IF MlegRollBFinished=FALSE AND (gait_cycle-EnterMlegRollBCount)<=MlegRollBTime*gvl.sampleRate THEN
	body_ref_pos:=body_ref_pos_enter;
	body_ref_ang:=body_ref_ang_enter;
	leg_ref_pos:=leg_ref_pos_enter;
	tr  := UDINT_TO_LREAL(gait_cycle - EnterMlegRollBCount) / gvl.sampleRate / MlegRollBTime;
	fbGetPivot(tNow := tr, tTotal := 1.0, pivot => pvt);
	FOR i:=0 TO 1 DO
		FOR j:=0 TO 2 DO
			MlegRollB_MJntRef[i].data[j]:=(1-pvt)*MlegRollB_MJntStart[i].data[j]+pvt*(MlegRollB_MJntTarget[i,j]);
		END_FOR
		gvl.legCtrl[Mapping14[i]].ForwardKinetics(motorAngles:=MlegRollB_MJntRef[i].data , legIndex:=Mapping14[i] , tipPosition=>MlegRollB_MPosWrtHip[i].data );
		fbRotMat(yaw := body_ref_ang_enter.data[2], pitch := body_ref_ang_enter.data[1],roll := body_ref_ang_enter.data[0], rm =>  Rb_target1 );
		temp.data[0]:=hip_pos[Mapping14[i],0];temp.data[1]:=hip_pos[Mapping14[i],1];temp.data[2]:=hip_pos[Mapping14[i],2];
		leg_ref_pos[Mapping14[i]]:= VecAdd( MatMulVec(Rb_target1, VecAdd(temp,MatMulVec(Rleg[Mapping14[i]],MlegRollB_MPosWrtHip[i]))),body_ref_pos);
	END_FOR
	
	//force compensator
	tipForceTarget:=tipForceDesireLegAF;
	IF (gait_cycle-EnterMlegRollBCount)<=fceLoadTime*gvl.sampleRate THEN
		tr  := UDINT_TO_LREAL(gait_cycle-EnterMlegRollBCount) / gvl.sampleRate / fceLoadTime;
		fbGetPivot(tNow := tr, tTotal := 1.0, pivot => pvt);
		FOR i:=0 TO 5 DO
			FOR j:=0 TO 2 DO
				tipForceDesire[i,j]:=(1-pvt)*tipForceDesireZeros[i,j]+pvt*tipForceTarget[i,j];
			END_FOR
		END_FOR
	ELSIF (gait_cycle-EnterMlegRollBCount)>(MlegRollBTime-fceLoadTime)*gvl.sampleRate AND (gait_cycle-EnterMlegRollBCount)<=MlegRollBTime*gvl.sampleRate THEN
		tr  := (UDINT_TO_LREAL(gait_cycle-EnterMlegRollBCount) / gvl.sampleRate -(MlegRollBTime-fceLoadTime))/ fceLoadTime;
		fbGetPivot(tNow := tr, tTotal := 1.0, pivot => pvt);
		FOR i:=0 TO 5 DO
			FOR j:=0 TO 2 DO
				tipForceDesire[i,j]:=(1-pvt)*tipForceTarget[i,j]+pvt*tipForceDesireZeros[i,j];
			END_FOR
		END_FOR	
	END_IF	
	
ELSE	
	MlegRollBFinished:=TRUE;
	tipForceDesire:=tipForceDesireZeros;
END_IF
END_METHOD

METHOD PUBLIC TrjPlanning_MlegRollC : BOOL
VAR_INPUT
END_VAR
VAR
	MlegRollC_MPosTarget:ARRAY[0..1,0..2] OF LREAL:=[-0.2,-0.1797,-0.1246,
                                                     -0.2,-0.1797,0.1246];
	MlegRollC_MJntTargetRef:ARRAY[0..1,0..2] OF LREAL:=[0,523.2736*pi/180,-235.1052*pi/180,
                                                     0,523.2736*pi/180,-235.1052*pi/180];//invert rotation for shank and thigh, a more rotation for shank, old version										 
													 
	tr: lreal;
	i: INT;
	j: INT;
	Rb_target1: Mat3;
	temp: vec3;
	tempLeg:ARRAY [0..2] OF LREAL;
	tempJnt:ARRAY [0..2] OF LREAL;
	tempRef:ARRAY [0..2] OF LREAL;	
	
	tipForceDesireLegAF:	 ARRAY[0..5,0..2] OF LREAL:=[0,-100,0,
													 0,0,0,
													 0,0,0,
													 0,0,0,
													 0,0,0,
													 0,-120,0];
END_VAR
IF (gait_cycle-EnterMlegRollCCount)=1 THEN
	FOR i:=0 TO 1 DO
		tempLeg[0]:=MlegRollC_MPosTarget[i,0];tempLeg[1]:=MlegRollC_MPosTarget[i,1];tempLeg[2]:=MlegRollC_MPosTarget[i,2];
		tempRef[0]:=MlegRollC_MJntTargetRef[i,0];tempRef[1]:=MlegRollC_MJntTargetRef[i,1];tempRef[2]:=MlegRollC_MJntTargetRef[i,2];
		GVL.legCtrl[Mapping14[i]].InverseKinetics(tipPosition:=tempLeg , refPosLast:=tempRef , legIndex:=Mapping14[i] , motorAngles=>tempJnt , isSingular=> );
		MlegRollC_MJntTarget[i,0]:=tempJnt[0];MlegRollC_MJntTarget[i,1]:=tempJnt[1];MlegRollC_MJntTarget[i,2]:=tempJnt[2];		
	END_FOR
END_IF

IF MlegRollCFinished=FALSE AND (gait_cycle-EnterMlegRollCCount)<=MlegRollCTime*gvl.sampleRate THEN
	body_ref_pos:=body_ref_pos_enter;
	body_ref_ang:=body_ref_ang_enter;
	leg_ref_pos:=leg_ref_pos_enter;
	
	tr  := UDINT_TO_LREAL(gait_cycle - EnterMlegRollCCount) / gvl.sampleRate / MlegRollCTime;
	fbGetPivot(tNow := tr, tTotal := 1.0, pivot => pvt);
	FOR i:=0 TO 1 DO
		FOR j:=0 TO 2 DO
			MlegRollC_MJntRef[i].data[j]:=(1-pvt)*MlegRollC_MJntStart[i].data[j]+pvt*(MlegRollC_MJntTarget[i,j]);
		END_FOR
		gvl.legCtrl[Mapping14[i]].ForwardKinetics(motorAngles:=MlegRollC_MJntRef[i].data , legIndex:=Mapping14[i] , tipPosition=>MlegRollC_MPosWrtHip[i].data );
		fbRotMat(yaw := body_ref_ang_enter.data[2], pitch := body_ref_ang_enter.data[1],roll := body_ref_ang_enter.data[0], rm =>  Rb_target1 );
		temp.data[0]:=hip_pos[Mapping14[i],0];temp.data[1]:=hip_pos[Mapping14[i],1];temp.data[2]:=hip_pos[Mapping14[i],2];
		leg_ref_pos[Mapping14[i]]:= VecAdd( MatMulVec(Rb_target1, VecAdd(temp,MatMulVec(Rleg[Mapping14[i]],MlegRollC_MPosWrtHip[i]))),body_ref_pos);
	END_FOR	
	
	//force compensator
	tipForceTarget:=tipForceDesireLegAF;
	IF (gait_cycle-EnterMlegRollCCount)<=fceLoadTime*gvl.sampleRate THEN
		tr  := UDINT_TO_LREAL(gait_cycle-EnterMlegRollCCount) / gvl.sampleRate / fceLoadTime;
		fbGetPivot(tNow := tr, tTotal := 1.0, pivot => pvt);
		FOR i:=0 TO 5 DO
			FOR j:=0 TO 2 DO
				tipForceDesire[i,j]:=(1-pvt)*tipForceDesireZeros[i,j]+pvt*tipForceTarget[i,j];
			END_FOR
		END_FOR
	ELSIF (gait_cycle-EnterMlegRollCCount)>(MlegRollCTime-fceLoadTime)*gvl.sampleRate AND (gait_cycle-EnterMlegRollCCount)<=MlegRollCTime*gvl.sampleRate THEN
		tr  := (UDINT_TO_LREAL(gait_cycle-EnterMlegRollCCount) / gvl.sampleRate -(MlegRollCTime-fceLoadTime))/ fceLoadTime;
		fbGetPivot(tNow := tr, tTotal := 1.0, pivot => pvt);
		FOR i:=0 TO 5 DO
			FOR j:=0 TO 2 DO
				tipForceDesire[i,j]:=(1-pvt)*tipForceTarget[i,j]+pvt*tipForceDesireZeros[i,j];
			END_FOR
		END_FOR	
	END_IF
	
ELSE	
	MlegRollCFinished:=TRUE;
	tipForceDesire:=tipForceDesireZeros;
	RequireAddHeight:=TRUE;//*******************************************************************************************************
END_IF
END_METHOD

METHOD PUBLIC TrjPlanning_OrientAdjust : BOOL
VAR_INPUT
END_VAR

VAR
	tr: LREAL;
	i: INT;
	Rb_target1: Mat3;
	temp: VEC3;
	j: INT;
	(*OA_MJntExtend:ARRAY[0..1,0..2] OF LREAL:=[0,331.45*pi/180,-144*pi/180,
                                                     0,331.45*pi/180,-144*pi/180];
	OA_MJntExtract:ARRAY[0..1,0..2] OF LREAL:=[0,340*pi/180,-155*pi/180,
                                                     0,340*pi/180,-155*pi/180];*)
END_VAR
IF OrientAdjustFinished=FALSE AND (gait_cycle-EnterOrientAdjustCount)<=LREAL_TO_UDINT((2*OA_LiftGroundTime+OA_AdjustTime+OA_AdjustExtractTime+OA_AdjustExtendTime)*gvl.sampleRate) THEN
	IF (gait_cycle-EnterOrientAdjustCount)<=LREAL_TO_UDINT((OA_LiftGroundTime)*gvl.sampleRate) THEN
		leg_ref_pos:=leg_ref_pos_enter;
		body_ref_ang:=OA_BodyAngStart;
		body_ref_pos:=OA_BodyPosStart;
		tr  := UDINT_TO_LREAL(gait_cycle - EnterOrientAdjustCount) / gvl.sampleRate /OA_LiftGroundTime;
		fbGetPivot(tNow := tr, tTotal := 1.0, pivot => pvt);	
		body_ref_pos.data[2]:=(1-pvt)*OA_BodyPosStart.data[2]+pvt*(OA_BodyPosStart.data[2]+OA_HeighAdd);
		FOR i:=0 TO 1 DO
			gvl.legCtrl[Mapping23[i]].ForwardKinetics(motorAngles:=OA_FJntRef[i].data , legIndex:=Mapping23[i] , tipPosition=>OA_FPosWrtHip[i].data );
			fbRotMat(yaw := body_ref_ang.data[2], pitch := body_ref_ang.data[1],roll := body_ref_ang.data[0], rm =>  Rb_target1 );
			temp.data[0]:=hip_pos[Mapping23[i],0];temp.data[1]:=hip_pos[Mapping23[i],1];temp.data[2]:=hip_pos[Mapping23[i],2];
			leg_ref_pos[Mapping23[i]]:= VecAdd( MatMulVec(Rb_target1, VecAdd(temp,MatMulVec(Rleg[Mapping23[i]],OA_FPosWrtHip[i]))),body_ref_pos);			
		END_FOR
	ELSIF (gait_cycle-EnterOrientAdjustCount)<=LREAL_TO_UDINT((OA_LiftGroundTime+OA_AdjustTime)*gvl.sampleRate) THEN
		leg_ref_pos:=leg_ref_pos_enter;
		tr  := (UDINT_TO_LREAL(gait_cycle - EnterOrientAdjustCount) / gvl.sampleRate -OA_LiftGroundTime)/OA_AdjustTime;
		fbGetPivot(tNow := tr, tTotal := 1.0, pivot => pvt);
		FOR i:=0 TO 2 DO
			body_ref_pos.data[i]:=(1-pvt)*OA_BodyPosStart.data[i]+pvt*OA_BodyPoseEnd.data[i];
			body_ref_ang.data[i]:=(1-pvt)*OA_BodyAngStart.data[i]+pvt*OA_BodyAngEnd.data[i];
		END_FOR		
		body_ref_pos.data[2]:=body_ref_pos.data[2]+OA_HeighAdd;
		FOR i:=0 TO 1 DO
			gvl.legCtrl[Mapping23[i]].ForwardKinetics(motorAngles:=OA_FJntRef[i].data , legIndex:=Mapping23[i] , tipPosition=>OA_FPosWrtHip[i].data );
			fbRotMat(yaw := body_ref_ang.data[2], pitch := body_ref_ang.data[1],roll := body_ref_ang.data[0], rm =>  Rb_target1 );
			temp.data[0]:=hip_pos[Mapping23[i],0];temp.data[1]:=hip_pos[Mapping23[i],1];temp.data[2]:=hip_pos[Mapping23[i],2];
			leg_ref_pos[Mapping23[i]]:= VecAdd( MatMulVec(Rb_target1, VecAdd(temp,MatMulVec(Rleg[Mapping23[i]],OA_FPosWrtHip[i]))),body_ref_pos);			
		END_FOR
	ELSIF (gait_cycle-EnterOrientAdjustCount)<=LREAL_TO_UDINT((2*OA_LiftGroundTime+OA_AdjustTime)*gvl.sampleRate) THEN	
		leg_ref_pos:=leg_ref_pos_enter;
		body_ref_ang:=OA_BodyAngEnd;
		body_ref_pos:=OA_BodyPoseEnd;
		tr  := (UDINT_TO_LREAL(gait_cycle - EnterOrientAdjustCount) / gvl.sampleRate-OA_LiftGroundTime-OA_AdjustTime )/OA_LiftGroundTime;
		fbGetPivot(tNow := tr, tTotal := 1.0, pivot => pvt);	
		body_ref_pos.data[2]:=(1-pvt)*(OA_BodyPosStart.data[2]+OA_HeighAdd)+pvt*OA_BodyPosStart.data[2];
		FOR i:=0 TO 1 DO
			gvl.legCtrl[Mapping23[i]].ForwardKinetics(motorAngles:=OA_FJntRef[i].data , legIndex:=Mapping23[i] , tipPosition=>OA_FPosWrtHip[i].data );
			fbRotMat(yaw := body_ref_ang.data[2], pitch := body_ref_ang.data[1],roll := body_ref_ang.data[0], rm =>  Rb_target1 );
			temp.data[0]:=hip_pos[Mapping23[i],0];temp.data[1]:=hip_pos[Mapping23[i],1];temp.data[2]:=hip_pos[Mapping23[i],2];
			leg_ref_pos[Mapping23[i]]:= VecAdd( MatMulVec(Rb_target1, VecAdd(temp,MatMulVec(Rleg[Mapping23[i]],OA_FPosWrtHip[i]))),body_ref_pos);			
		END_FOR		
		IF (gait_cycle-EnterOrientAdjustCount)=LREAL_TO_UDINT((2*OA_LiftGroundTime+OA_AdjustTime)*gvl.sampleRate) THEN
			OA_legPosEnterExtract:=leg_ref_pos;
			FOR i:=0 TO 1 DO
				FOR j:=0 TO 2 DO
					OA_MJntStart[i].data[j]:=jointPosLast[Mapping14[i],j];
				END_FOR
			END_FOR			
		END_IF
	ELSIF (gait_cycle-EnterOrientAdjustCount)<=LREAL_TO_UDINT((2*OA_LiftGroundTime+OA_AdjustTime+OA_AdjustExtractTime)*gvl.sampleRate) THEN	
		body_ref_pos:=OA_BodyPoseEnd;
		body_ref_ang:=OA_BodyAngEnd;
		leg_ref_pos:=OA_legPosEnterExtract;
		tr  := (UDINT_TO_LREAL(gait_cycle - EnterOrientAdjustCount) / gvl.sampleRate-2*OA_LiftGroundTime-OA_AdjustTime )/OA_AdjustExtractTime;
		fbGetPivot(tNow := tr, tTotal := 1.0, pivot => pvt);	
		FOR i:=0 TO 1 DO
			FOR j:=0 TO 2 DO
				OA_MJntRef[i].data[j]:=(1-pvt)*OA_MJntStart[i].data[j]+pvt*OA_MJntExtract[i,j];
			END_FOR
			gvl.legCtrl[Mapping14[i]].ForwardKinetics(motorAngles:=OA_MJntRef[i].data , legIndex:=Mapping14[i] , tipPosition=>OA_MPosWrtHip[i].data );
			fbRotMat(yaw := body_ref_ang.data[2], pitch := body_ref_ang.data[1],roll := body_ref_ang.data[0], rm =>  Rb_target1 );
			temp.data[0]:=hip_pos[Mapping14[i],0];temp.data[1]:=hip_pos[Mapping14[i],1];temp.data[2]:=hip_pos[Mapping14[i],2];
			leg_ref_pos[Mapping14[i]]:= VecAdd( MatMulVec(Rb_target1, VecAdd(temp,MatMulVec(Rleg[Mapping14[i]],OA_MPosWrtHip[i]))),body_ref_pos);
			
			gvl.legCtrl[Mapping23[i]].ForwardKinetics(motorAngles:=OA_FJntRef[i].data , legIndex:=Mapping23[i] , tipPosition=>OA_FPosWrtHip[i].data );
			temp.data[0]:=hip_pos[Mapping23[i],0];temp.data[1]:=hip_pos[Mapping23[i],1];temp.data[2]:=hip_pos[Mapping23[i],2];
			leg_ref_pos[Mapping23[i]]:= VecAdd( MatMulVec(Rb_target1, VecAdd(temp,MatMulVec(Rleg[Mapping23[i]],OA_FPosWrtHip[i]))),body_ref_pos);	
		END_FOR		
	ELSE
		body_ref_pos:=OA_BodyPoseEnd;
		body_ref_ang:=OA_BodyAngEnd;
		leg_ref_pos:=OA_legPosEnterExtract;	
		tr  := (UDINT_TO_LREAL(gait_cycle - EnterOrientAdjustCount) / gvl.sampleRate-2*OA_LiftGroundTime-OA_AdjustTime-OA_AdjustExtractTime )/OA_AdjustExtendTime;
		fbGetPivot(tNow := tr, tTotal := 1.0, pivot => pvt);
		FOR i:=0 TO 1 DO
			FOR j:=0 TO 2 DO
				OA_MJntRef[i].data[j]:=(1-pvt)*OA_MJntExtract[i,j]+pvt*OA_MJntExtend[i,j];
			END_FOR		
			gvl.legCtrl[Mapping14[i]].ForwardKinetics(motorAngles:=OA_MJntRef[i].data , legIndex:=Mapping14[i] , tipPosition=>OA_MPosWrtHip[i].data );
			fbRotMat(yaw := body_ref_ang.data[2], pitch := body_ref_ang.data[1],roll := body_ref_ang.data[0], rm =>  Rb_target1 );
			temp.data[0]:=hip_pos[Mapping14[i],0];temp.data[1]:=hip_pos[Mapping14[i],1];temp.data[2]:=hip_pos[Mapping14[i],2];
			leg_ref_pos[Mapping14[i]]:= VecAdd( MatMulVec(Rb_target1, VecAdd(temp,MatMulVec(Rleg[Mapping14[i]],OA_MPosWrtHip[i]))),body_ref_pos);	

			gvl.legCtrl[Mapping23[i]].ForwardKinetics(motorAngles:=OA_FJntRef[i].data , legIndex:=Mapping23[i] , tipPosition=>OA_FPosWrtHip[i].data );
			temp.data[0]:=hip_pos[Mapping23[i],0];temp.data[1]:=hip_pos[Mapping23[i],1];temp.data[2]:=hip_pos[Mapping23[i],2];
			leg_ref_pos[Mapping23[i]]:= VecAdd( MatMulVec(Rb_target1, VecAdd(temp,MatMulVec(Rleg[Mapping23[i]],OA_FPosWrtHip[i]))),body_ref_pos);		
		END_FOR					
	END_IF
ELSE
	OrientAdjustFinished:=TRUE;
END_IF
END_METHOD

METHOD PUBLIC TrjPlanning_PushReleaseBall : BOOL
VAR_INPUT
END_VAR

VAR
	PushReleaseBall_FJntTarget:ARRAY[0..1,0..2] OF LREAL:=[-90*pi/180,155*pi/180,175*pi/180,
                                                     90*pi/180,155*pi/180,175*pi/180];//prepared position before gripping stone													 
													 
	i,j: INT;
	invalid: LREAL;
	Rb_target1: Mat3;
	temp: vec3;
	flag: INT;
	tr: LREAL;
END_VAR
//push and release method
IF PushReleaseBallFinished=FALSE AND gvl.curlingPushModel=0 THEN
	body_ref_pos:=body_ref_pos_enter;
	body_ref_ang:=body_ref_ang_enter;
	leg_ref_pos:=leg_ref_pos_enter;
	FOR i:=0 TO 1 DO
		IF gait_cycle-EnterPushReleaseBallCount<=PushTime*gvl.sampleRate THEN
			fbHermitInterpolation(t0:=EnterPushReleaseBallCount*delta_t , T:=PushTime , y0:=PushReleaseBall_FPosStartWrtHip[i].data[0] , 
			y1:=PushReleaseBall_FPosStartWrtHip[i].data[0]-PushDistance , v0:=0 , v1:=-PushVelocity , tNow:=(gait_cycle)* delta_t, 
			y=> PushReleaseBall_FPosWrtHip[i].data[0], v=>invalid );
		ELSIF gait_cycle-EnterPushReleaseBallCount<=(PushTime+PRConstVelTime)*gvl.sampleRate THEN
			fbHermitInterpolation(t0:=EnterPushReleaseBallCount*delta_t+PushTime , T:=PRConstVelTime , y0:=PushReleaseBall_FPosStartWrtHip[i].data[0]-PushDistance , 
			y1:=PushReleaseBall_FPosStartWrtHip[i].data[0]-PushDistance-PRConstVelDistance , v0:=-PushVelocity , v1:= -PushVelocity, tNow:=gait_cycle* delta_t, 
			y=> PushReleaseBall_FPosWrtHip[i].data[0], v=>invalid );			
		ELSIF gait_cycle-EnterPushReleaseBallCount<=(PushTime+PRConstVelTime+DecVelTime)*gvl.sampleRate THEN
			fbHermitInterpolation(t0:=EnterPushReleaseBallCount*delta_t+PushTime+PRConstVelTime , T:=DecVelTime , y0:=PushReleaseBall_FPosStartWrtHip[i].data[0]-PushDistance-PRConstVelDistance , 
			y1:=PushReleaseBall_FPosStartWrtHip[i].data[0]-PushDistance-PRConstVelDistance-DecVelDistance , v0:=-PushVelocity , v1:= 0, tNow:=gait_cycle* delta_t, 
			y=> PushReleaseBall_FPosWrtHip[i].data[0], v=>invalid );	
		ELSE
			 PushReleaseBall_FPosWrtHip[i].data[0]:=PushReleaseBall_FPosStartWrtHip[i].data[0]-PushDistance-PRConstVelDistance-DecVelDistance;	
			 PushReleaseBallFinished:=TRUE;	
			 EnterPushFinishCount:=gait_cycle;
			 
		END_IF
		PushReleaseBall_FPosWrtHip[i].data[1]:=PushReleaseBall_FPosStartWrtHip[i].data[1];
		PushReleaseBall_FPosWrtHip[i].data[2]:=PushReleaseBall_FPosStartWrtHip[i].data[2];
		
		fbRotMat(yaw := body_ref_ang_enter.data[2], pitch := body_ref_ang_enter.data[1],roll := body_ref_ang_enter.data[0], rm =>  Rb_target1 );
		temp.data[0]:=hip_pos[Mapping23[i],0];temp.data[1]:=hip_pos[Mapping23[i],1];temp.data[2]:=hip_pos[Mapping23[i],2];
		leg_ref_pos[Mapping23[i]]:= VecAdd( MatMulVec(Rb_target1, VecAdd(temp,MatMulVec(Rleg[Mapping23[i]],PushReleaseBall_FPosWrtHip[i]))),body_ref_pos);
	END_FOR
END_IF



//only release method
IF PushReleaseBallFinished=FALSE AND gvl.curlingPushModel=1 THEN
	IF gait_cycle - EnterPushReleaseBallCount<=ReleaseTime*gvl.sampleRate THEN
		body_ref_pos:=body_ref_pos_enter;
		body_ref_ang:=body_ref_ang_enter;
		leg_ref_pos:=leg_ref_pos_enter;
	
		tr  := UDINT_TO_LREAL(gait_cycle - EnterPushReleaseBallCount) / gvl.sampleRate / ReleaseTime;
		fbGetPivot(tNow := tr, tTotal := 1.0, pivot => pvt);
		FOR i:=0 TO 1 DO
			FOR j:=0 TO 2 DO
				PushReleaseBall_FJntRef[i].data[j]:=(1-pvt)*PushReleaseBall_FJntStart[i].data[j]+pvt*(PushReleaseBall_FJntTarget[i,j]);
			END_FOR
			gvl.legCtrl[Mapping23[i]].ForwardKinetics(motorAngles:=PushReleaseBall_FJntRef[i].data , legIndex:=Mapping23[i] , tipPosition=>PushReleaseBall_FPosWrtHip[i].data );
			fbRotMat(yaw := body_ref_ang_enter.data[2], pitch := body_ref_ang_enter.data[1],roll := body_ref_ang_enter.data[0], rm =>  Rb_target1 );
			temp.data[0]:=hip_pos[Mapping23[i],0];temp.data[1]:=hip_pos[Mapping23[i],1];temp.data[2]:=hip_pos[Mapping23[i],2];
			leg_ref_pos[Mapping23[i]]:= VecAdd( MatMulVec(Rb_target1, VecAdd(temp,MatMulVec(Rleg[Mapping23[i]],PushReleaseBall_FPosWrtHip[i]))),body_ref_pos);
		END_FOR
	ELSE	
		PushReleaseBallFinished:=TRUE;
		EnterPushFinishCount:=gait_cycle;
	END_IF	
END_IF

IF PushReleaseBallFinished=TRUE AND SpeedDownFinished=FALSE AND gait_cycle-EnterPushFinishCount>=LREAL_TO_UDINT(PushFinishDurationTime)*gvl.sampleRate  THEN
	RequireSpeedDown:=TRUE;
END_IF
END_METHOD

METHOD PUBLIC TrjPlanning_Recovery : BOOL
VAR_INPUT
END_VAR
VAR
	legExtractRefPosCurling: ARRAY[0..5, 0..2] OF LREAL:=[-0.35,-0.3+0.02,0,
														  0.1,-0.3+0.02,-0.1246,
														  -0.15,-0.3+0.02,-0.1246,
														  -0.15,-0.3+0.02,0.1246,
														  0.1,-0.3+0.02,0.1246,
														  -0.35,-0.3+0.02,0];
	jntExtractRefPosCurling: ARRAY[0..5, 0..2] OF LREAL:=[0,163.1808*pi/180,297.208*pi/180,
											  			  0,322.9120*pi/180,(205.1705-322.9120)*pi/180,
											              0,183.8227*pi/180,(269.8634-183.8227)*pi/180,
											              0,183.8227*pi/180,(269.8634-183.8227)*pi/180,
											              0,322.9120*pi/180,(205.1705-322.9120)*pi/180,
											              0,163.1808*pi/180,297.208*pi/180];
	legExtendRefPosCurling: ARRAY[0..5, 0..2] OF LREAL:=[-0.35,-0.4-0.07,0,
														  0.1,-0.4-0.07,-0.1246,
														  -0.15,-0.4-0.07,-0.1246,
														  -0.15,-0.4-0.07,0.1246,
														  0.1,-0.4-0.07,0.1246,
														  -0.35,-0.4-0.07,0];														 
	jntExtendRefPosCurling: ARRAY[0..5, 0..2] OF LREAL:=[0,181.9845*pi/180,299.9603*pi/180,
											 			 0,302.7132*pi/180,(230.9946-302.7132)*pi/180,	
											             0,222.0252*pi/180,(254.0072-222.0252)*pi/180,
											             0,222.0252*pi/180,(254.0072-222.0252)*pi/180,
									                     0,302.7132*pi/180,(230.9946-302.7132)*pi/180,
											             0,181.9845*pi/180,299.9603*pi/180]	;

	(*legExtractRefPosCurling:    ARRAY[0..5, 0..2] OF LREAL:=[-0.35,-0.3+0.08,0,
														  0.1,-0.3209+0.08,-0.1246,
														  -0.3,-0.3209+0.08,-0.1246,
														  -0.3,-0.3209+0.08,0.1246,
														  0.1,-0.3209+0.08,0.1246,
														  -0.35,-0.3+0.08,0];															  
	jntExtractRefPosCurling: ARRAY[0..5, 0..2] OF LREAL:= [0,150.7997*pi/180,291.8958*pi/180,
											  			0,327.8142*pi/180,(196.8366-327.8142)*pi/180,
											  			0,172.5134*pi/180,(269.4767-172.5134)*pi/180,
											  			0,172.5134*pi/180,(269.4767-172.5134)*pi/180,
											  			0,327.8142*pi/180,(196.8366-327.8142)*pi/180,
											  			0,150.7997*pi/180,291.8958*pi/180];	
	legExtendRefPosCurling: ARRAY[0..5, 0..2] OF LREAL    :=[-0.35,-0.3209,0,
														  0.1,-0.3209,-0.1246,
														  -0.3,-0.3209,-0.1246,
														  -0.3,-0.3209,0.1246,
														  0.1,-0.3209,0.1246,
														  -0.35,-0.3209,0];														  													  
	jntExtendRefPosCurling: ARRAY[0..5, 0..2] OF LREAL:=	[0,163.1808*pi/180,297.208*pi/180,
											 				0,320.9331*pi/180,(208.0880-320.9331)*pi/180,	
											 				0,187.8384*pi/180,(269.4264-187.8384)*pi/180,
															0,187.8384*pi/180,(269.4264-187.8384)*pi/180,
									         				0,320.9331*pi/180,(208.0880-320.9331)*pi/180,
											 				0,163.1808*pi/180,297.208*pi/180];*)
													  
	i: INT;
	j: INT;
	tempLeg:ARRAY [0..2] OF LREAL;
	tempJnt:ARRAY [0..2] OF LREAL;
	tempRef:ARRAY [0..2] OF LREAL;
	tTotal: LREAL;
	tNow: LREAL;
	jntPosBegin : ARRAY[0..5, 0..2] OF LREAL;
	jntPosEnd   : ARRAY[0..5, 0..2] OF LREAL;
	Rb_target1: Mat3;
	temp: vec3;
	tipForceDesireGroupA:ARRAY[0..5,0..2] OF LREAL:=[0,-100,0,
													 0,0,0,
													 0,0,0,
													 0,0,0,
													 0,0,0,
													 0,0,0];
	tipForceDesireGroupB:ARRAY[0..5,0..2] OF LREAL:=[0,0,0,
													 0,0,0,
													 0,0,0,
													 0,0,0,
													 0,0,0,
													 0,-120,0];
	tr: LREAL;
END_VAR
IF (gait_cycle-EnterRecoveryCount)=1 THEN
	FOR i:=0 TO 5 DO
		tempLeg[0]:=legExtractRefPosCurling[i,0];tempLeg[1]:=legExtractRefPosCurling[i,1];tempLeg[2]:=legExtractRefPosCurling[i,2];
		tempRef[0]:=jntExtractRefPosCurling[i,0];tempRef[1]:=jntExtractRefPosCurling[i,1];tempRef[2]:=jntExtractRefPosCurling[i,2];
		GVL.legCtrl[i].InverseKinetics(tipPosition:=tempLeg , refPosLast:=tempRef , legIndex:=i , motorAngles=>tempJnt , isSingular=> );
		jntAngRetract[i,0]:=tempJnt[0];jntAngRetract[i,1]:=tempJnt[1];jntAngRetract[i,2]:=tempJnt[2];
		
		tempLeg[0]:=legExtendRefPosCurling[i,0];tempLeg[1]:=legExtendRefPosCurling[i,1];tempLeg[2]:=legExtendRefPosCurling[i,2];
		tempRef[0]:=jntExtendRefPosCurling[i,0];tempRef[1]:=jntExtendRefPosCurling[i,1];tempRef[2]:=jntExtendRefPosCurling[i,2];
		GVL.legCtrl[i].InverseKinetics(tipPosition:=tempLeg , refPosLast:=tempRef , legIndex:=i , motorAngles=>tempJnt , isSingular=> );
		jntAngExtend[i,0]:=tempJnt[0];jntAngExtend[i,1]:=tempJnt[1];jntAngExtend[i,2]:=tempJnt[2];			
		
	END_FOR
	tipForceDesire:=tipForceDesireZeros;

END_IF

IF RecoveryFinished=FALSE THEN
	body_ref_pos:=body_ref_pos_enter;
	body_ref_ang:=body_ref_ang_enter;
	leg_ref_pos:=leg_ref_pos_enter;
	
	IF (gait_cycle-EnterRecoveryCount)<=(tRetract + tWait + tExtend) * gvl.sampleRate THEN //leg 0-2-4 recovery
		
		//force compensator****************************
		IF (gait_cycle-EnterRecoveryCount)<=fceLoadTime*gvl.sampleRate THEN
			tr  := UDINT_TO_LREAL(gait_cycle-EnterRecoveryCount) / gvl.sampleRate /fceLoadTime;
			fbGetPivot(tNow := tr, tTotal := 1.0, pivot => pvt);
			FOR i:=0 TO 5 DO
				FOR j:=0 TO 2 DO
					tipForceDesire[i,j]:=(1-pvt)*tipForceDesireZeros[i,j]+pvt*tipForceDesireGroupB[i,j];//group B add load
				END_FOR
			END_FOR
		ELSIF  (gait_cycle-EnterRecoveryCount)>LREAL_TO_UDINT((tRetract + tWait + tExtend-fceLoadTime)*gvl.sampleRate) AND  (gait_cycle-EnterRecoveryCount)<=LREAL_TO_UDINT((tRetract + tWait + tExtend) * gvl.sampleRate) THEN
			tr  := (UDINT_TO_LREAL (gait_cycle-EnterRecoveryCount) / gvl.sampleRate-(tRetract + tWait + tExtend-fceLoadTime) )/fceLoadTime;
			fbGetPivot(tNow := tr, tTotal := 1.0, pivot => pvt);
			FOR i:=0 TO 5 BY 2DO
				FOR j:=0 TO 2 DO
					//tipForceDesire[i,j]:=(1-pvt)*tipForceDesireZeros[i,j]+pvt*tipForceDesireGroupA[i,j];//group A add load
					tipForceDesire[i+1,j]:=(1-pvt)*tipForceDesireGroupB[i+1,j]+pvt*tipForceDesireZeros[i+1,j];//group B reduce load
				END_FOR
			END_FOR
		ELSE
		tipForceDesire:=tipForceDesireGroupB;
		END_IF
		//***********************************************
	
		IF gait_cycle-EnterRecoveryCount < tRetract * gvl.sampleRate THEN
			tTotal := tRetract;
			tNow   := UDINT_TO_LREAL(gait_cycle-EnterRecoveryCount) * 1.0 / DINT_TO_LREAL(gvl.sampleRate);
			jntPosBegin := RcJointPosStart;
			FOR i:=0 TO 5 BY 2 DO
				FOR j:=0 TO 2 DO
					jntPosEnd[i,j]:=jntAngRetract[i,j];
					jntPosEnd[i+1,j]:=RcJointPosStart[i+1,j];
				END_FOR
			END_FOR
		ELSIF gait_cycle-EnterRecoveryCount  < (tRetract + tWait) * gvl.sampleRate THEN
			tTotal := tWait;
			tNow   := UDINT_TO_LREAL(gait_cycle-EnterRecoveryCount) * 1.0 / DINT_TO_LREAL(gvl.sampleRate) - tRetract;
			FOR i:=0 TO 5 BY 2 DO
				FOR j:=0 TO 2 DO
					jntPosBegin[i,j]:=jntAngRetract[i,j];
					jntPosBegin[i+1,j]:=RcJointPosStart[i+1,j];
					jntPosEnd[i,j]:=jntAngRetract[i,j];
					jntPosEnd[i+1,j]:=RcJointPosStart[i+1,j];
				END_FOR
			END_FOR
		ELSE 
			tTotal := tExtend;
			tNow   := UDINT_TO_LREAL(gait_cycle-EnterRecoveryCount) * 1.0 / DINT_TO_LREAL(gvl.sampleRate) - tRetract - tWait;
			FOR i:=0 TO 5 BY 2 DO
				FOR j:=0 TO 2 DO
					jntPosBegin[i,j]:=jntAngRetract[i,j];
					jntPosBegin[i+1,j]:=RcJointPosStart[i+1,j];
					jntPosEnd[i,j]:=jntAngExtend[i,j];
					jntPosEnd[i+1,j]:=RcJointPosStart[i+1,j];
				END_FOR
			END_FOR	
		END_IF	
	ELSIF (gait_cycle-EnterRecoveryCount)<=2*(tRetract + tWait + tExtend) * gvl.sampleRate  THEN //leg 1-3-5 recovery

		//force compensator*******************
		IF (gait_cycle-EnterRecoveryCount)>LREAL_TO_UDINT((tRetract + tWait + tExtend)*gvl.sampleRate) AND (gait_cycle-EnterRecoveryCount)<=LREAL_TO_UDINT((tRetract + tWait + tExtend+fceLoadTime)* gvl.sampleRate) THEN
			tr  := (UDINT_TO_LREAL(gait_cycle-EnterRecoveryCount) / gvl.sampleRate-(tRetract + tWait + tExtend) )/fceLoadTime;
			fbGetPivot(tNow := tr, tTotal := 1.0, pivot => pvt);
			FOR i:=0 TO 5 BY 2 DO
				FOR j:=0 TO 2 DO
					tipForceDesire[i,j]:=(1-pvt)*tipForceDesireZeros[i,j]+pvt*tipForceDesireGroupA[i,j];//group A add load
					tipForceDesire[i+1,j]:=tipForceDesireZeros[i+1,j];//group B zeros load
				END_FOR
			END_FOR		
		ELSIF (gait_cycle-EnterRecoveryCount)>LREAL_TO_UDINT((2*(tRetract + tWait + tExtend)-fceLoadTime)*gvl.sampleRate) AND (gait_cycle-EnterRecoveryCount)<=LREAL_TO_UDINT(2*(tRetract + tWait + tExtend) * gvl.sampleRate) THEN
			tr  := (UDINT_TO_LREAL(gait_cycle-EnterRecoveryCount) / gvl.sampleRate-(2*(tRetract + tWait + tExtend)-fceLoadTime) )/fceLoadTime;
			fbGetPivot(tNow := tr, tTotal := 1.0, pivot => pvt);
			FOR i:=0 TO 5 BY 2DO
				FOR j:=0 TO 2 DO
					tipForceDesire[i,j]:=(1-pvt)*tipForceDesireGroupA[i,j]+pvt*tipForceDesireZeros[i,j];//group A reduce load
					tipForceDesire[i+1,j]:=tipForceDesireZeros[i+1,j];//group B zeros load
				END_FOR
			END_FOR	
		ELSE	
			tipForceDesire:=tipForceDesireGroupA;
		END_IF	
		//******************************************	

		
		IF gait_cycle-EnterRecoveryCount<=(2*tRetract + tWait + tExtend) * gvl.sampleRate THEN
			tTotal := tRetract;
			tNow   := UDINT_TO_LREAL(gait_cycle-EnterRecoveryCount) * 1.0 / DINT_TO_LREAL(gvl.sampleRate)-(tRetract + tWait + tExtend);
			FOR i:=0 TO 5 BY 2 DO
				FOR j:=0 TO 2 DO
					jntPosBegin[i,j]:=jntAngExtend[i,j];
					jntPosBegin[i+1,j]:=RcJointPosStart[i+1,j];
					jntPosEnd[i,j]:=jntAngExtend[i,j];
					jntPosEnd[i+1,j]:=jntAngRetract[i+1,j];
				END_FOR
			END_FOR			
		ELSIF gait_cycle-EnterRecoveryCount<=(2*tRetract + 2*tWait + tExtend) * gvl.sampleRate THEN
			tTotal := tWait;
			tNow   := UDINT_TO_LREAL(gait_cycle-EnterRecoveryCount) * 1.0 / DINT_TO_LREAL(gvl.sampleRate) - (2*tRetract + tWait + tExtend);
			FOR i:=0 TO 5 BY 2 DO
				FOR j:=0 TO 2 DO
					jntPosBegin[i,j]:=jntAngExtend[i,j];
					jntPosBegin[i+1,j]:=jntAngRetract[i+1,j];
					jntPosEnd[i,j]:=jntAngExtend[i,j];
					jntPosEnd[i+1,j]:=jntAngRetract[i+1,j];
				END_FOR
			END_FOR			
		ELSE
			tTotal := tExtend;
			tNow   := UDINT_TO_LREAL(gait_cycle-EnterRecoveryCount) * 1.0 / DINT_TO_LREAL(gvl.sampleRate) - (2*tRetract + 2*tWait + tExtend);
			FOR i:=0 TO 5 BY 2 DO
				FOR j:=0 TO 2 DO
					jntPosBegin[i,j]:=jntAngExtend[i,j];
					jntPosBegin[i+1,j]:=jntAngRetract[i+1,j];
					jntPosEnd[i,j]:=jntAngExtend[i,j];
					jntPosEnd[i+1,j]:=jntAngExtend[i+1,j];
				END_FOR
			END_FOR			
		END_IF
	ELSE
		tTotal := 100;
		tNow   := UDINT_TO_LREAL(gait_cycle-EnterRecoveryCount) * 1.0 / DINT_TO_LREAL(gvl.sampleRate) - 2*tRetract - 2*tWait - 2*tExtend;
		jntPosBegin :=jntAngExtend;
		jntPosEnd :=jntAngExtend;
		RecoveryFinished:=TRUE;
		tipForceDesire:=tipForceDesireZeros;
	END_IF
	getPivot(tNow := tNow, tTotal := tTotal, pivot => pivot, pivotDot => pivotDot);
	FOR i := 0 TO 5 DO
		FOR j := 0 TO 2 DO
			RcJointPosRef[i, j] := (1.0 - pivot) * jntPosBegin[i, j] + pivot * jntPosEnd[i, j];
		END_FOR
		tempJnt[0]:=RcJointPosRef[i,0];tempJnt[1]:=RcJointPosRef[i,1];tempJnt[2]:=RcJointPosRef[i,2];
		gvl.legCtrl[i].ForwardKinetics(motorAngles:=tempJnt , legIndex:=i , tipPosition=>Rc_PosWrtHip[i].data );
		fbRotMat(yaw := body_ref_ang_enter.data[2], pitch := body_ref_ang_enter.data[1],roll := body_ref_ang_enter.data[0], rm =>  Rb_target1 );
		temp.data[0]:=hip_pos[i,0];temp.data[1]:=hip_pos[i,1];temp.data[2]:=hip_pos[i,2];
		leg_ref_pos[i]:= VecAdd( MatMulVec(Rb_target1, VecAdd(temp,MatMulVec(Rleg[i],Rc_PosWrtHip[i]))),body_ref_pos);		
	END_FOR

END_IF
END_METHOD

METHOD PUBLIC TrjPlanning_ReduceHeight : BOOL
VAR_INPUT
	
END_VAR
VAR
	
	tr: LREAL;
	i: INT;
	Rb_target1: Mat3;
	temp: vec3;
END_VAR
IF ReduceHeightFinished=FALSE AND (gait_cycle-EnterReduceHeightCount)<=ReduceHeightTime*gvl.sampleRate THEN
	body_ref_ang:=body_ref_ang_enter;
	leg_ref_pos:=leg_ref_pos_enter;
	tr  := UDINT_TO_LREAL(gait_cycle - EnterReduceHeightCount) / gvl.sampleRate / ReduceHeightTime;
	fbGetPivot(tNow := tr, tTotal := 1.0, pivot => pvt);
	FOR i:=0 TO 2 DO
		body_ref_pos.data[i]:=(1-pvt)*body_ref_pos_enter.data[i]+pvt*body_target_pos.data[i];
	END_FOR
	FOR i:=0 TO 1 DO
		gvl.legCtrl[Mapping23[i]].ForwardKinetics(motorAngles:=ReduceHeight_FJntRef[i].data , legIndex:=Mapping23[i] , tipPosition=>ReduceHeight_FPosWrtHip[i].data );
		fbRotMat(yaw := body_ref_ang_enter.data[2], pitch := body_ref_ang_enter.data[1],roll := body_ref_ang_enter.data[0], rm =>  Rb_target1 );
		temp.data[0]:=hip_pos[Mapping23[i],0];temp.data[1]:=hip_pos[Mapping23[i],1];temp.data[2]:=hip_pos[Mapping23[i],2];
		leg_ref_pos[Mapping23[i]]:= VecAdd( MatMulVec(Rb_target1, VecAdd(temp,MatMulVec(Rleg[Mapping23[i]],ReduceHeight_FPosWrtHip[i]))),body_ref_pos);
	END_FOR
ELSE
	ReduceHeightFinished:=TRUE;
END_IF
END_METHOD

METHOD PUBLIC TrjPlanning_SearchPedal : BOOL
VAR_INPUT
END_VAR
VAR
	tr: LREAL;
	i: INT;
	j: INT;
	Rb_target1: Mat3;
	temp: vec3;
	
	tipForceDesireLegA:	 ARRAY[0..5,0..2] OF LREAL:=[0,-100,0,
													 0,0,0,
													 0,0,0,
													 0,0,0,
													 0,0,0,
													 0,0,0];
	tipForceDesireLegF:	 ARRAY[0..5,0..2] OF LREAL:=[0,0,0,
													 0,0,0,
													 0,0,0,
													 0,0,0,
													 0,0,0,
													 0,-120,0];				
END_VAR
IF SearchPedalFinished=FALSE THEN
	IF SP_RBLegSearching=TRUE THEN
		SP_LBLegSearching:=FALSE;
		body_ref_pos:=body_ref_pos_enter;
		body_ref_ang:=body_ref_ang_enter;
		leg_ref_pos:=leg_ref_pos_enter;	
		IF (gait_cycle-SP_EnterSubSearchCount[0])<=SP_LiftLegTime*gvl.sampleRate THEN
			tr  := UDINT_TO_LREAL(gait_cycle - SP_EnterSubSearchCount[0]) / gvl.sampleRate / SP_LiftLegTime;
			fbGetPivot(tNow := tr, tTotal := 1.0, pivot => pvt);	
			SP_BPosRefWrtHip[0].data[0]:=SP_BPosStartWrtHip[0].data[0];
			SP_BPosRefWrtHip[0].data[1]:=(1-pvt)*SP_BPosStartWrtHip[0].data[1]+pvt*(SP_BPosStartWrtHip[0].data[1]+SP_LiftDistance);
			SP_BPosRefWrtHip[0].data[2]:=SP_BPosStartWrtHip[0].data[2];
			fbRotMat(yaw := body_ref_ang_enter.data[2], pitch := body_ref_ang_enter.data[1],roll := body_ref_ang_enter.data[0], rm =>  Rb_target1 );
			temp.data[0]:=hip_pos[0,0];temp.data[1]:=hip_pos[0,1];temp.data[2]:=hip_pos[0,2];
			leg_ref_pos[0]:= VecAdd( MatMulVec(Rb_target1, VecAdd(temp,MatMulVec(Rleg[0],SP_BPosRefWrtHip[0]))),body_ref_pos);	
			
			//force compensator
			tipForceTarget:=tipForceDesireLegF;
			IF (gait_cycle-SP_EnterSubSearchCount[0])<=LREAL_TO_UDINT(fceLoadTime*gvl.sampleRate) THEN
				tr  := (UDINT_TO_LREAL(gait_cycle-SP_EnterSubSearchCount[0]) / gvl.sampleRate)/ fceLoadTime;
				fbGetPivot(tNow := tr, tTotal := 1.0, pivot => pvt);
				FOR i:=0 TO 5 DO
					FOR j:=0 TO 2 DO
						tipForceDesire[i,j]:=(1-pvt)*tipForceDesireZeros[i,j]+pvt*tipForceTarget[i,j];
					END_FOR
				END_FOR
			END_IF
			
		ELSIF (gait_cycle-SP_EnterSubSearchCount[0])<=(SP_LiftLegTime+SP_SearchTime)*gvl.sampleRate AND  SP_BLegSearchFinished[0]=FALSE THEN
			tr  := (UDINT_TO_LREAL(gait_cycle - SP_EnterSubSearchCount[0]) / gvl.sampleRate -SP_LiftLegTime)/ SP_SearchTime;
			fbGetPivot(tNow := tr, tTotal := 1.0, pivot => pvt);	
			SP_BPosRefWrtHip[0].data[0]:=(1-pvt)*SP_BPosStartWrtHip[0].data[0]+pvt*(SP_BPosStartWrtHip[0].data[0]-SP_SearchDistance);		
			SP_BPosRefWrtHip[0].data[1]:=SP_BPosStartWrtHip[0].data[1]+SP_LiftDistance;
			SP_BPosRefWrtHip[0].data[2]:=SP_BPosStartWrtHip[0].data[2];
			IF isPedal(0)=TRUE AND  SP_BLegSearchFinished[0]=FALSE THEN
				SP_BLegSearchFinished[0]:=TRUE;
				SP_EnterSubSearchDecreaseCount[0]:=gait_cycle;
				FOR j:=0 TO 2 DO
					SP_BPosLockWrtHip[0].data[j]:=SP_BPosRefWrtHip[0].data[j];
				END_FOR			
			END_IF
			IF (gait_cycle-SP_EnterSubSearchCount[0])=LREAL_TO_UDINT((SP_LiftLegTime+SP_SearchTime)*gvl.sampleRate) AND SP_BLegSearchFinished[0]=FALSE THEN
				SP_BLegSearchFinished[0]:=TRUE;
				SP_EnterSubSearchDecreaseCount[0]:=gait_cycle;
				FOR j:=0 TO 2 DO
					SP_BPosLockWrtHip[0].data[j]:=SP_BPosRefWrtHip[0].data[j];
				END_FOR	
			END_IF

			fbRotMat(yaw := body_ref_ang_enter.data[2], pitch := body_ref_ang_enter.data[1],roll := body_ref_ang_enter.data[0], rm =>  Rb_target1 );
			temp.data[0]:=hip_pos[0,0];temp.data[1]:=hip_pos[0,1];temp.data[2]:=hip_pos[0,2];
			leg_ref_pos[0]:= VecAdd( MatMulVec(Rb_target1, VecAdd(temp,MatMulVec(Rleg[0],SP_BPosRefWrtHip[0]))),body_ref_pos);	
			
		ELSIF  SP_BLegSearchFinished[0]=TRUE AND (gait_cycle-SP_EnterSubSearchDecreaseCount[0])<=SP_LiftLegTime*gvl.sampleRate THEN
			tr  := UDINT_TO_LREAL(gait_cycle - SP_EnterSubSearchDecreaseCount[0]) / gvl.sampleRate / SP_LiftLegTime;
			fbGetPivot(tNow := tr, tTotal := 1.0, pivot => pvt);
			SP_BPosRefWrtHip[0].data[0]:=SP_BPosLockWrtHip[0].data[0];	
			SP_BPosRefWrtHip[0].data[1]:=(1-pvt)*SP_BPosLockWrtHip[0].data[1]+pvt*(SP_BPosLockWrtHip[0].data[1]-SP_LiftDistance);
			SP_BPosRefWrtHip[0].data[2]:=SP_BPosLockWrtHip[0].data[2];	
			
			fbRotMat(yaw := body_ref_ang_enter.data[2], pitch := body_ref_ang_enter.data[1],roll := body_ref_ang_enter.data[0], rm =>  Rb_target1 );
			temp.data[0]:=hip_pos[0,0];temp.data[1]:=hip_pos[0,1];temp.data[2]:=hip_pos[0,2];
			leg_ref_pos[0]:= VecAdd( MatMulVec(Rb_target1, VecAdd(temp,MatMulVec(Rleg[0],SP_BPosRefWrtHip[0]))),body_ref_pos);	
			IF (gait_cycle-SP_EnterSubSearchDecreaseCount[0])=LREAL_TO_UDINT( SP_LiftLegTime*gvl.sampleRate) THEN
				body_ref_pos_enter:=body_ref_pos;
				body_ref_ang_enter:=body_ref_ang;
				leg_ref_pos_enter:=leg_ref_pos;	
			END_IF	
			
			//force compensator
			tipForceTarget:=tipForceDesireLegF;
			IF (gait_cycle-SP_EnterSubSearchDecreaseCount[0])>LREAL_TO_UDINT((SP_LiftLegTime-fceLoadTime)*gvl.sampleRate)THEN
				tr  := (UDINT_TO_LREAL(gait_cycle-SP_EnterSubSearchDecreaseCount[0]) / gvl.sampleRate-(SP_LiftLegTime-fceLoadTime) )/ fceLoadTime;
				fbGetPivot(tNow := tr, tTotal := 1.0, pivot => pvt);
				FOR i:=0 TO 5 DO
					FOR j:=0 TO 2 DO
						tipForceDesire[i,j]:=(1-pvt)*tipForceTarget[i,j]+pvt*tipForceDesireZeros[i,j];
					END_FOR
				END_FOR
			END_IF
	
		ELSE
			SP_RBLegSearching:=FALSE;
			SP_LBLegSearching:=TRUE;
			SP_EnterSubSearchCount[1]:=gait_cycle;			
		END_IF
	END_IF
	
	IF SP_LBLegSearching=TRUE THEN
		SP_RBLegSearching:=FALSE;
		body_ref_pos:=body_ref_pos_enter;
		body_ref_ang:=body_ref_ang_enter;
		leg_ref_pos:=leg_ref_pos_enter;	
		IF (gait_cycle-SP_EnterSubSearchCount[1])<=SP_LiftLegTime*gvl.sampleRate THEN
			tr  := UDINT_TO_LREAL(gait_cycle - SP_EnterSubSearchCount[1]) / gvl.sampleRate / SP_LiftLegTime;
			fbGetPivot(tNow := tr, tTotal := 1.0, pivot => pvt);	
			SP_BPosRefWrtHip[1].data[0]:=SP_BPosStartWrtHip[1].data[0];
			SP_BPosRefWrtHip[1].data[1]:=(1-pvt)*SP_BPosStartWrtHip[1].data[1]+pvt*(SP_BPosStartWrtHip[1].data[1]+SP_LiftDistance);
			SP_BPosRefWrtHip[1].data[2]:=SP_BPosStartWrtHip[1].data[2];
			fbRotMat(yaw := body_ref_ang_enter.data[2], pitch := body_ref_ang_enter.data[1],roll := body_ref_ang_enter.data[0], rm =>  Rb_target1 );
			temp.data[0]:=hip_pos[5,0];temp.data[1]:=hip_pos[5,1];temp.data[2]:=hip_pos[5,2];
			leg_ref_pos[5]:= VecAdd( MatMulVec(Rb_target1, VecAdd(temp,MatMulVec(Rleg[5],SP_BPosRefWrtHip[1]))),body_ref_pos);	
			
			//force compensator
			tipForceTarget:=tipForceDesireLegA;
			IF (gait_cycle-SP_EnterSubSearchCount[1])<=LREAL_TO_UDINT(fceLoadTime*gvl.sampleRate) THEN
				tr  := (UDINT_TO_LREAL(gait_cycle-SP_EnterSubSearchCount[1]) / gvl.sampleRate)/ fceLoadTime;
				fbGetPivot(tNow := tr, tTotal := 1.0, pivot => pvt);
				FOR i:=0 TO 5 DO
					FOR j:=0 TO 2 DO
						tipForceDesire[i,j]:=(1-pvt)*tipForceDesireZeros[i,j]+pvt*tipForceTarget[i,j];
					END_FOR
				END_FOR
			END_IF
			
		ELSIF (gait_cycle-SP_EnterSubSearchCount[1])<=(SP_LiftLegTime+SP_SearchTime)*gvl.sampleRate AND  SP_BLegSearchFinished[1]=FALSE THEN
			tr  := (UDINT_TO_LREAL(gait_cycle - SP_EnterSubSearchCount[1]) / gvl.sampleRate -SP_LiftLegTime)/ SP_SearchTime;
			fbGetPivot(tNow := tr, tTotal := 1.0, pivot => pvt);	
			SP_BPosRefWrtHip[1].data[0]:=(1-pvt)*SP_BPosStartWrtHip[1].data[0]+pvt*(SP_BPosStartWrtHip[1].data[0]-SP_SearchDistance);		
			SP_BPosRefWrtHip[1].data[1]:=SP_BPosStartWrtHip[1].data[1]+SP_LiftDistance;
			SP_BPosRefWrtHip[1].data[2]:=SP_BPosStartWrtHip[1].data[2];
			IF isPedal(5)=TRUE AND  SP_BLegSearchFinished[1]=FALSE THEN
				SP_BLegSearchFinished[1]:=TRUE;
				SP_EnterSubSearchDecreaseCount[1]:=gait_cycle;
				FOR j:=0 TO 2 DO
					SP_BPosLockWrtHip[1].data[j]:=SP_BPosRefWrtHip[1].data[j];
				END_FOR			
			END_IF
			IF (gait_cycle-SP_EnterSubSearchCount[1])=LREAL_TO_UDINT((SP_LiftLegTime+SP_SearchTime)*gvl.sampleRate) AND SP_BLegSearchFinished[1]=FALSE THEN
				SP_BLegSearchFinished[1]:=TRUE;
				SP_EnterSubSearchDecreaseCount[1]:=gait_cycle;
				FOR j:=0 TO 2 DO
					SP_BPosLockWrtHip[1].data[j]:=SP_BPosRefWrtHip[1].data[j];
				END_FOR	
			END_IF

			fbRotMat(yaw := body_ref_ang_enter.data[2], pitch := body_ref_ang_enter.data[1],roll := body_ref_ang_enter.data[0], rm =>  Rb_target1 );
			temp.data[0]:=hip_pos[5,0];temp.data[1]:=hip_pos[5,1];temp.data[2]:=hip_pos[5,2];
			leg_ref_pos[5]:= VecAdd( MatMulVec(Rb_target1, VecAdd(temp,MatMulVec(Rleg[5],SP_BPosRefWrtHip[1]))),body_ref_pos);	
			
		ELSIF  SP_BLegSearchFinished[1]=TRUE AND (gait_cycle-SP_EnterSubSearchDecreaseCount[1])<=SP_LiftLegTime*gvl.sampleRate THEN
			tr  := UDINT_TO_LREAL(gait_cycle - SP_EnterSubSearchDecreaseCount[1]) / gvl.sampleRate / SP_LiftLegTime;
			fbGetPivot(tNow := tr, tTotal := 1.0, pivot => pvt);
			SP_BPosRefWrtHip[1].data[0]:=SP_BPosLockWrtHip[1].data[0];	
			SP_BPosRefWrtHip[1].data[1]:=(1-pvt)*SP_BPosLockWrtHip[1].data[1]+pvt*(SP_BPosLockWrtHip[1].data[1]-SP_LiftDistance);
			SP_BPosRefWrtHip[1].data[2]:=SP_BPosLockWrtHip[1].data[2];	
			
			fbRotMat(yaw := body_ref_ang_enter.data[2], pitch := body_ref_ang_enter.data[1],roll := body_ref_ang_enter.data[0], rm =>  Rb_target1 );
			temp.data[0]:=hip_pos[5,0];temp.data[1]:=hip_pos[5,1];temp.data[2]:=hip_pos[5,2];
			leg_ref_pos[5]:= VecAdd( MatMulVec(Rb_target1, VecAdd(temp,MatMulVec(Rleg[5],SP_BPosRefWrtHip[1]))),body_ref_pos);	
			IF (gait_cycle-SP_EnterSubSearchDecreaseCount[1])=LREAL_TO_UDINT( SP_LiftLegTime*gvl.sampleRate) THEN
				body_ref_pos_enter:=body_ref_pos;
				body_ref_ang_enter:=body_ref_ang;
				leg_ref_pos_enter:=leg_ref_pos;	
			END_IF	
			
			//force compensator
			tipForceTarget:=tipForceDesireLegA;
			IF (gait_cycle-SP_EnterSubSearchDecreaseCount[1])>LREAL_TO_UDINT((SP_LiftLegTime-fceLoadTime)*gvl.sampleRate)THEN
				tr  := (UDINT_TO_LREAL(gait_cycle-SP_EnterSubSearchDecreaseCount[1]) / gvl.sampleRate-(SP_LiftLegTime-fceLoadTime) )/ fceLoadTime;
				fbGetPivot(tNow := tr, tTotal := 1.0, pivot => pvt);
				FOR i:=0 TO 5 DO
					FOR j:=0 TO 2 DO
						tipForceDesire[i,j]:=(1-pvt)*tipForceTarget[i,j]+pvt*tipForceDesireZeros[i,j];
					END_FOR
				END_FOR
			END_IF			
			
		ELSE
			SP_RBLegSearching:=FALSE;
			SP_LBLegSearching:=FALSE;	
			SearchPedalFinished:=TRUE;	
			tipForceDesire:=tipForceDesireZeros;
		END_IF
	END_IF	
END_IF
END_METHOD

METHOD PUBLIC TrjPlanning_Slide : BOOL
VAR_INPUT
END_VAR
IF SlideFinished=FALSE THEN
	body_ref_pos:=body_ref_pos_enter;
	body_ref_ang:=body_ref_ang_enter;
	leg_ref_pos:=leg_ref_pos_enter;

END_IF

//***********tuning***************************
IF SlideFinished=FALSE AND (gait_cycle-EnterSlideCount)>=LREAL_TO_UDINT(slideTime*gvl.sampleRate) THEN
	RequirePushReleaseBall:=TRUE;
END_IF

//*************end-tuning********************



IF SlideFinished=FALSE AND RequirePushReleaseBall=TRUE THEN
	SlideFinished:=TRUE;
END_IF
END_METHOD

METHOD PUBLIC TrjPlanning_SpeedDown : BOOL
VAR_INPUT
END_VAR

VAR
	tr: LREAL;
	i: INT;
	SpeedDown_MPosTarget:ARRAY[0..1,0..2] OF LREAL:=[-0.0141,-0.1797,-0.1246,
                                                        -0.0141,-0.1797,0.1246];
	SpeedDown_MJntTargetRef:ARRAY[0..1,0..2] OF LREAL:=[0,331.45*pi/180,-144*pi/180,
                                                     0,331.45*pi/180,-144*pi/180];
	j: INT;
	Rb_target1: Mat3;
	temp: vec3;
	tempLeg:ARRAY [0..2] OF LREAL;
	tempJnt:ARRAY [0..2] OF LREAL;
	tempRef:ARRAY [0..2] OF LREAL;
END_VAR
IF (gait_cycle-EnterSpeedDownCount)=1 THEN
	FOR i:=0 TO 1 DO
		tempLeg[0]:=SpeedDown_MPosTarget[i,0];tempLeg[1]:=SpeedDown_MPosTarget[i,1];tempLeg[2]:=SpeedDown_MPosTarget[i,2];
		tempRef[0]:=SpeedDown_MJntTargetRef[i,0];tempRef[1]:=SpeedDown_MJntTargetRef[i,1];tempRef[2]:=SpeedDown_MJntTargetRef[i,2];
		GVL.legCtrl[Mapping14[i]].InverseKinetics(tipPosition:=tempLeg , refPosLast:=tempRef , legIndex:=Mapping14[i] , motorAngles=>tempJnt , isSingular=> );
		SpeedDown_MJntTarget[i,0]:=tempJnt[0];SpeedDown_MJntTarget[i,1]:=tempJnt[1];SpeedDown_MJntTarget[i,2]:=tempJnt[2];		
	END_FOR
END_IF

IF SpeedDownFinished=FALSE THEN
	IF gait_cycle-EnterSpeedDownCount<=SpeedDownTime*gvl.sampleRate THEN
		body_ref_pos:=body_ref_pos_enter;
		body_ref_ang:=body_ref_ang_enter;
		leg_ref_pos:=leg_ref_pos_enter;
		tr  := UDINT_TO_LREAL(gait_cycle - EnterSpeedDownCount) / gvl.sampleRate / SpeedDownTime;
		fbGetPivot(tNow := tr, tTotal := 1.0, pivot => pvt);
		FOR i:=0 TO 1 DO
			FOR j:=0 TO 2 DO
				SpeedDown_MJntRef[i].data[j]:=(1-pvt)*SpeedDown_MJntStart[i].data[j]+pvt*SpeedDown_MJntTarget[i,j];
			END_FOR
			gvl.legCtrl[Mapping14[i]].ForwardKinetics(motorAngles:=SpeedDown_MJntRef[i].data , legIndex:=Mapping14[i] , tipPosition=>SpeedDown_MPosWrtHip[i].data );
			fbRotMat(yaw := body_ref_ang_enter.data[2], pitch := body_ref_ang_enter.data[1],roll := body_ref_ang_enter.data[0], rm =>  Rb_target1 );
			temp.data[0]:=hip_pos[Mapping14[i],0];temp.data[1]:=hip_pos[Mapping14[i],1];temp.data[2]:=hip_pos[Mapping14[i],2];
			leg_ref_pos[Mapping14[i]]:= VecAdd( MatMulVec(Rb_target1, VecAdd(temp,MatMulVec(Rleg[Mapping14[i]],SpeedDown_MPosWrtHip[i]))),body_ref_pos);
			
			leg_ref_pos[Mapping05[i]].data[2]:=(1-pvt)*leg_ref_pos_enter[Mapping05[i]].data[2]+pvt*(leg_ref_pos_enter[Mapping05[i]].data[2]-Distance_y_DS-0.005);
		END_FOR
	ELSE
		SpeedDownFinished:=TRUE;
		
	END_IF
	
	IF gait_cycle-EnterSpeedDownCount=1 THEN
		GVL.jogVelocity[18]:=0;
		GVL.jogVelocity[19]:=0;
		gvl.jogStopButton[18]:=TRUE;
		gvl.jogStopButton[19]:=TRUE;
		gvl.motorDrive[j].SetTrgVel(0);
	END_IF
END_IF
END_METHOD

METHOD PUBLIC TrjPlanning_SpeedUp : BOOL
VAR_INPUT
END_VAR

VAR
	invalid: LREAL;
	Rb_target1: Mat3;
	i: INT;
	tr: LREAL;
	temp: VEC3;
	
	
	tipForceDesireLegAF:	 ARRAY[0..5,0..2] OF LREAL:=[0,-5,0,
													 0,0,0,
													 0,0,0,
													 0,0,0,
													 0,0,0,
													 0,-5,0];
	j: INT;
END_VAR
IF SpeedUpSubState=SpeedUpAS AND (gait_cycle-EnterSpeedUpASCount)=LREAL_TO_UDINT(Time_AS*gvl.sampleRate) THEN
	SpeedUpSubState:=SpeedUpCS;
	EnterSpeedUpCSCount:=gait_cycle;
	body_ref_pos_enter :=body_ref_pos;
	body_ref_ang_enter:=body_ref_ang;
	leg_ref_pos_enter := leg_ref_pos;
	
ELSIF SpeedUpSubState=SpeedUpCS AND gait_cycle-EnterSpeedUpCSCount=LREAL_TO_UDINT(Time_CS*gvl.sampleRate) THEN
	SpeedUpSubState:=SpeedUpDS;
	EnterSpeedUpDSCount:=gait_cycle;
	body_ref_pos_enter :=body_ref_pos;
	body_ref_ang_enter:=body_ref_ang;
	leg_ref_pos_enter := leg_ref_pos;
ELSIF SpeedUpSubState=SpeedUpDS AND gait_cycle-EnterSpeedUpDSCount=LREAL_TO_UDINT(Time_DS*gvl.sampleRate) THEN
	SpeedUpSubState:=SpeedUpSS;
	EnterSpeedUpSPCount:=gait_cycle;
	body_ref_pos_enter :=body_ref_pos;
	body_ref_ang_enter:=body_ref_ang;
	leg_ref_pos_enter := leg_ref_pos;
	SpeedUpFinished:=TRUE;
	tipForceDesire:=tipForceDesireZeros;
	RequireSlide:=TRUE;
END_IF

body_ref_pos:=body_ref_pos_enter;
body_ref_ang:=body_ref_ang_enter;
leg_ref_pos:=leg_ref_pos_enter;

IF SpeedUpSubState=SpeedUpAS AND gait_cycle-EnterSpeedUpASCount<=Time_AS*gvl.sampleRate THEN
	fbHermitInterpolation(t0:=EnterSpeedUpASCount*delta_t , T:=Time_AS , y0:=0 , 
		y1:=Distance_x_AS , v0:=0 , v1:=target_vel , tNow:=gait_cycle* delta_t, 
		y=> body_ref_pos_wrt_body.data[0], v=>invalid );	
	body_ref_pos_wrt_body.data[1]:=0;body_ref_pos_wrt_body.data[2]:=0;
	fbRotMat(yaw := body_ref_ang_enter.data[2], pitch := body_ref_ang_enter.data[1],roll := body_ref_ang_enter.data[0], rm =>  Rb_target1 );
	body_ref_pos:=VecAdd(body_ref_pos_enter,MatMulVec(Rb_target1,body_ref_pos_wrt_body));
	
	//force compensator
	tipForceTarget:=tipForceDesireLegAF;
	IF (gait_cycle-EnterSpeedUpASCount)<=fceLoadTime*gvl.sampleRate THEN
		tr  := UDINT_TO_LREAL(gait_cycle-EnterSpeedUpASCount) / gvl.sampleRate / fceLoadTime;
		fbGetPivot(tNow := tr, tTotal := 1.0, pivot => pvt);
		FOR i:=0 TO 5 DO
			FOR j:=0 TO 2 DO
				tipForceDesire[i,j]:=(1-pvt)*tipForceDesireZeros[i,j]+pvt*tipForceTarget[i,j];
			END_FOR
		END_FOR	
	END_IF
	
END_IF
	//force compensator
	tipForceTarget:=tipForceDesireLegAF;
	IF (gait_cycle-EnterSpeedUpASCount)>(Time_AS+Time_CS-fceLoadTime)*gvl.sampleRate AND (gait_cycle-EnterSpeedUpASCount)<=(Time_AS+Time_CS)*gvl.sampleRate THEN
		tr  := (UDINT_TO_LREAL(gait_cycle-EnterSpeedUpASCount) / gvl.sampleRate- (Time_AS+Time_CS-fceLoadTime))/ fceLoadTime;
		fbGetPivot(tNow := tr, tTotal := 1.0, pivot => pvt);
		FOR i:=0 TO 5 DO
			FOR j:=0 TO 2 DO
				tipForceDesire[i,j]:=(1-pvt)*tipForceTarget[i,j]+pvt*tipForceDesireZeros[i,j];
			END_FOR
		END_FOR	
	END_IF

IF SpeedUpSubState=SpeedUpCS AND gait_cycle-EnterSpeedUpCSCount<=Time_CS*gvl.sampleRate THEN
	fbHermitInterpolation(t0:=EnterSpeedUpCSCount*delta_t , T:=Time_CS , y0:=0 , 
		y1:=target_vel*Time_CS , v0:=target_vel , v1:=target_vel , tNow:=gait_cycle* delta_t, 
		y=> body_ref_pos_wrt_body.data[0], v=>invalid );
	body_ref_pos_wrt_body.data[1]:=0;body_ref_pos_wrt_body.data[2]:=0;
	fbRotMat(yaw := body_ref_ang_enter.data[2], pitch := body_ref_ang_enter.data[1],roll := body_ref_ang_enter.data[0], rm =>  Rb_target1 );
	body_ref_pos:=VecAdd(body_ref_pos_enter,MatMulVec(Rb_target1,body_ref_pos_wrt_body));
END_IF
IF SpeedUpSubState=SpeedUpDS AND gait_cycle-EnterSpeedUpDSCount<=Time_DS*gvl.sampleRate THEN
	fbHermitInterpolation(t0:=EnterSpeedUpDSCount*delta_t , T:=Time_DS , y0:=0 , 
		y1:=Distance_x_DS , v0:=target_vel , v1:=0 , tNow:=gait_cycle* delta_t, 
		y=> body_ref_pos_wrt_body.data[0], v=>invalid );
	body_ref_pos_wrt_body.data[1]:=0;body_ref_pos_wrt_body.data[2]:=0;
	
	fbRotMat(yaw := body_ref_ang_enter.data[2], pitch := body_ref_ang_enter.data[1],roll := body_ref_ang_enter.data[0], rm =>  Rb_target1 );
	body_ref_pos:=VecAdd(body_ref_pos_enter,MatMulVec(Rb_target1,body_ref_pos_wrt_body));
	
	tr  := UDINT_TO_LREAL(gait_cycle - EnterSpeedUpDSCount) / gvl.sampleRate / Time_DS;
	fbGetPivot(tNow := tr, tTotal := 1.0, pivot => pvt);
	FOR i:=0 TO 1 DO
		leg_ref_pos[Mapping05[i]].data[2]:=(1-pvt)*leg_ref_pos_enter[Mapping05[i]].data[2]+pvt*(leg_ref_pos_enter[Mapping05[i]].data[2]+Distance_y_DS);
	END_FOR
	
END_IF
IF SpeedUpSubState=SpeedUpAS OR SpeedUpSubState=SpeedUpCS OR SpeedUpSubState=SpeedUpDS THEN
	FOR i:=0 TO 1 DO
		gvl.legCtrl[Mapping14[i]].ForwardKinetics(motorAngles:=SpeedUp_MJntRef[i].data , legIndex:=Mapping14[i] , tipPosition=>SpeedUp_MPosWrtHip[i].data );
		gvl.legCtrl[Mapping23[i]].ForwardKinetics(motorAngles:=SpeedUp_FJntRef[i].data , legIndex:=Mapping23[i] , tipPosition=>SpeedUp_FPosWrtHip[i].data );
		fbRotMat(yaw := body_ref_ang_enter.data[2], pitch := body_ref_ang_enter.data[1],roll := body_ref_ang_enter.data[0], rm =>  Rb_target1 );
		temp.data[0]:=hip_pos[Mapping14[i],0];temp.data[1]:=hip_pos[Mapping14[i],1];temp.data[2]:=hip_pos[Mapping14[i],2];
		leg_ref_pos[Mapping14[i]]:= VecAdd( MatMulVec(Rb_target1, VecAdd(temp,MatMulVec(Rleg[Mapping14[i]],SpeedUp_MPosWrtHip[i]))),body_ref_pos);
		temp.data[0]:=hip_pos[Mapping23[i],0];temp.data[1]:=hip_pos[Mapping23[i],1];temp.data[2]:=hip_pos[Mapping23[i],2];
		leg_ref_pos[Mapping23[i]]:= VecAdd( MatMulVec(Rb_target1, VecAdd(temp,MatMulVec(Rleg[Mapping23[i]],SpeedUp_FPosWrtHip[i]))),body_ref_pos);
	END_FOR
END_IF
END_METHOD

METHOD PUBLIC TrjPlanning_StoneRot : BOOL
VAR_INPUT
END_VAR
VAR
	(*StoneRot_FJntTarget:ARRAY[0..1,0..2] OF LREAL:=[-90*pi/180,524*pi/180,-190*pi/180,
                                                     90*pi/180,524*pi/180,-190*pi/180];*)
													 
	(*StoneRot_FJntTarget:ARRAY[0..1,0..2] OF LREAL:=[-90*pi/180,165*pi/180,(-190+360)*pi/180,
                                                     90*pi/180,165*pi/180,(-190+360)*pi/180];	//164 lose,165T 170S lose;*)
	StoneRot_FJntTarget:ARRAY[0..1,0..2] OF LREAL:=[-90*pi/180,167*pi/180,(171)*pi/180,
                                                     90*pi/180,167*pi/180,(171)*pi/180];	//164 lose,166T 168S passive wheels colide;												 
	tr: LREAL;
	i: INT;
	Rb_target1: Mat3;	
	temp:vec3;										 
	j: INT;
	noPlanning: BOOL;
END_VAR
//*****************************test trajectory*****************************************

	FOR i:=0 TO 1 DO
		(*IF SetColide=TRUE THEN
			gvl.tipActualFce[Mapping23[i],2]:=100;
		END_IF	*)
		(*IF(gait_cycle-EnterStoneRotCount)=0.5*StoneGripTime*gvl.sampleRate THEN
			gvl.tipActualFce[Mapping23[i],2]:=100;
		END_IF *)
		noPlanning:=TRUE;
	END_FOR
	

//**********************************end************************************************	

(*FOR i:=0 TO 1 DO
	IF StoneRotSubState[i]=FALSE AND isStone(Mapping23[i]) THEN
		StoneRotSubState[i]:=TRUE;
		leg_ref_pos_enter[Mapping23[i]]:=leg_ref_pos[Mapping23[i]];
	END_IF
END_FOR*)

IF (StoneRotSubState[0]=FALSE OR StoneRotSubState[1]=FALSE) AND (gait_cycle-EnterStoneRotCount)=LREAL_TO_UDINT(StoneGripTime*gvl.sampleRate) THEN
	StoneRotSubState[0]:=TRUE;
	StoneRotSubState[1]:=TRUE;
	leg_ref_pos_enter[Mapping23[0]]:=leg_ref_pos[Mapping23[0]];
	leg_ref_pos_enter[Mapping23[1]]:=leg_ref_pos[Mapping23[1]];
END_IF
	
body_ref_pos:=body_ref_pos_enter;
body_ref_ang:=body_ref_ang_enter;
leg_ref_pos:=leg_ref_pos_enter;


	IF (gait_cycle-EnterStoneRotCount)<=StoneGripTime*gvl.sampleRate THEN
		FOR i:=0 TO 1 DO
			IF StoneRotSubState[i]=FALSE THEN
			tr  := UDINT_TO_LREAL(gait_cycle - EnterStoneRotCount) / gvl.sampleRate /StoneGripTime;
			fbGetPivot(tNow := tr, tTotal := 1.0, pivot => pvt);
			FOR j:=0 TO 2 DO
				StoneRot_FJntRef[i].data[j]:=(1-pvt)*StoneRot_FJntStart[i].data[j]+pvt*(StoneRot_FJntTarget[i,j]);
			END_FOR
			gvl.legCtrl[Mapping23[i]].ForwardKinetics(motorAngles:=StoneRot_FJntRef[i].data , legIndex:=Mapping23[i] , tipPosition=>StoneRot_FPosWrtHip[i].data );
			fbRotMat(yaw := body_ref_ang_enter.data[2], pitch := body_ref_ang_enter.data[1],roll := body_ref_ang_enter.data[0], rm =>  Rb_target1 );
			temp.data[0]:=hip_pos[Mapping23[i],0];temp.data[1]:=hip_pos[Mapping23[i],1];temp.data[2]:=hip_pos[Mapping23[i],2];
			leg_ref_pos[Mapping23[i]]:= VecAdd( MatMulVec(Rb_target1, VecAdd(temp,MatMulVec(Rleg[Mapping23[i]],StoneRot_FPosWrtHip[i]))),body_ref_pos);
			END_IF
		END_FOR
	ELSE
		noPlanning:=TRUE;
	END_IF

IF (gait_cycle-EnterStoneRotCount)>StoneGripTime*gvl.sampleRate  THEN
		stone_rot_vel:=GVL.stone_rot_vel/60*2*pi;
		GVL.jogVelocity[18]:=stone_rot_vel;
		GVL.jogVelocity[19]:=-stone_rot_vel;
		FOR j:=18 TO 19 DO
			gvl.motorDrive[j].SetTrgVel(GVL.jogVelocity[j]);
			IF gvl.motorDrive[j].cvSetVel = GVL.jogVelocity[j] THEN
				gvl.jogButton[j]:=FALSE;
			ELSE
				gvl.jogButton[j]:=TRUE;
			END_IF
		END_FOR
END_IF

IF StoneRotFinished=FALSE AND (gait_cycle-EnterStoneRotCount)>=(StoneGripTime+StoneRotTime)*gvl.sampleRate THEN
	StoneRotFinished:=TRUE;
END_IF
END_METHOD

END_FUNCTION_BLOCK

(* stored: Version 1.1.0.1, ProductVersion 3.1.4024.2
   POU CurlingGaitFromStance: Id {d0604e6f-9105-4b2c-95cd-a4548dedf4a6}, SpecialFunc None
   Method DoPlanning: Id {8911b8c7-48bc-4012-aef3-3a58d43d6c47}
   Method Initialize: Id {24766bc0-7e6c-41f1-add8-e0d633233b90}
   Method isPedal: Id {93926f98-ae8f-4076-ab0f-a8bbdb4b82d2}
   Method isStone: Id {9ca69fac-a946-4015-9412-c595289bd6c1}
   Method SetTargetValue: Id {aa3b189f-f971-484c-91e4-923cd6060880}
   Method StateMachine: Id {f4aa490d-cb90-4397-b1a5-d47a080970e0}
   Method TrjPlanning: Id {2c06c156-67b3-4507-b886-ced2e376c983}
   Method TrjPlanning_AddHeight: Id {b2dc6c77-2d57-4310-88d3-24284b5db998}
   Method TrjPlanning_ArmControl: Id {23b87d45-09cd-46a8-af31-20409c836d92}
   Method TrjPlanning_BlegCenter: Id {f3dde1d6-0958-429c-9551-6848441a7774}
   Method TrjPlanning_BLegPosAdjust: Id {89eff12d-d682-4133-92c8-02c331bc91e3}
   Method TrjPlanning_BLegRecovery: Id {7c1a42fe-a4a8-4a4e-a2b1-2257c5078686}
   Method TrjPlanning_BodyPosAdjust: Id {f66f26aa-d130-4291-9e30-b1d5a24bc6c3}
   Method TrjPlanning_FlegRotA: Id {154d9726-17ea-437f-b24d-531f477e8a47}
   Method TrjPlanning_FlegRotB: Id {586665da-5f6e-40eb-b875-13ac50d1a40a}
   Method TrjPlanning_LiftMleg: Id {5219b450-f32e-4634-a8dd-4253d51b6f22}
   Method TrjPlanning_MlegRollA: Id {a49dfe94-0389-402a-b402-722171139aeb}
   Method TrjPlanning_MlegRollB: Id {43841e6f-f59b-48d1-be78-6a8e553953af}
   Method TrjPlanning_MlegRollC: Id {6482210e-6c83-4407-bacf-de2e57af19bf}
   Method TrjPlanning_OrientAdjust: Id {f582601e-4f11-41e5-8288-b8030d059854}
   Method TrjPlanning_PushReleaseBall: Id {f79100c5-363f-42a3-9118-ec9492481d3c}
   Method TrjPlanning_Recovery: Id {2db8ccc5-f9fe-4bc9-b9cf-67d331424a77}
   Method TrjPlanning_ReduceHeight: Id {398e25d4-1a05-4919-a3fc-1255f2862a99}
   Method TrjPlanning_SearchPedal: Id {6e7ce6ff-6be3-465d-9a84-48a1ac58dc4a}
   Method TrjPlanning_Slide: Id {9d695c40-fb36-4da4-84dc-7782aabb993b}
   Method TrjPlanning_SpeedDown: Id {e2631118-c6c0-4297-88b4-fcd6debd523a}
   Method TrjPlanning_SpeedUp: Id {79688172-18ab-4f41-9f12-e156878ca017}
   Method TrjPlanning_StoneRot: Id {1424996b-8c76-4ceb-83bd-a7216b9c72e2} *)
